# B&R Automation Studio project Lab2_Conveyor (part 4)

### Program Logical/Sorting/AlarmCtrl (IEC) - Alarm control for sorter

#### Cyclic.ld - Cyclic code
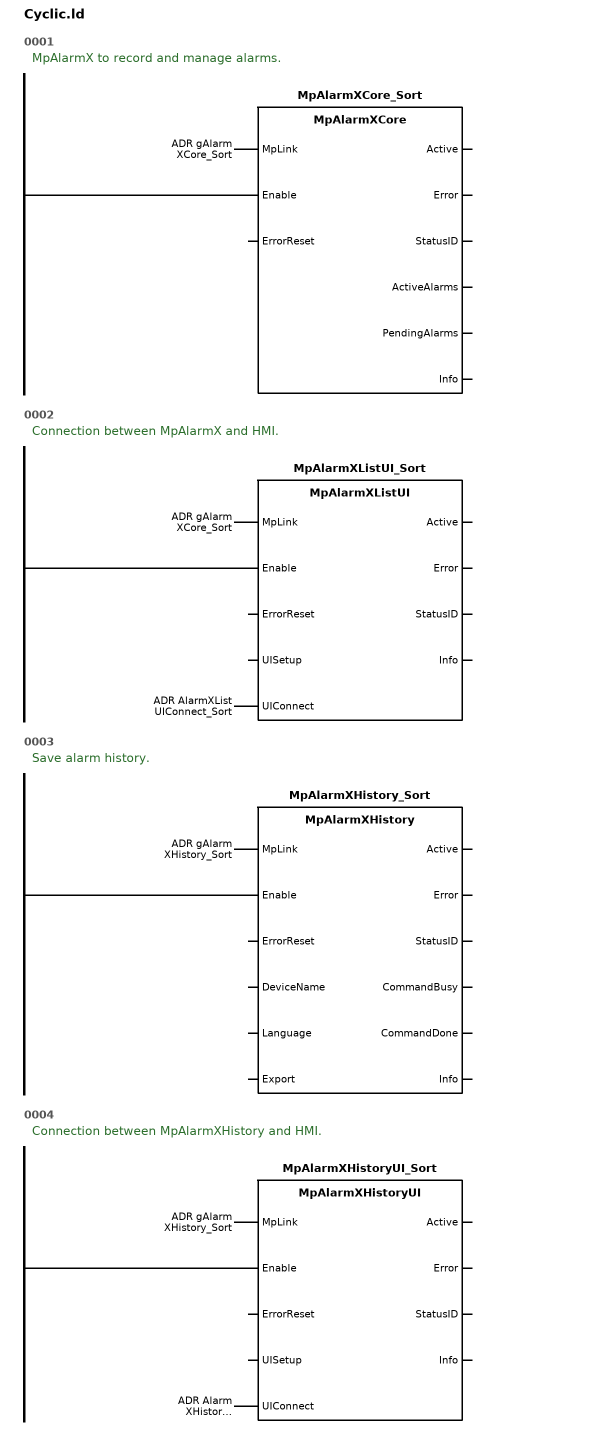
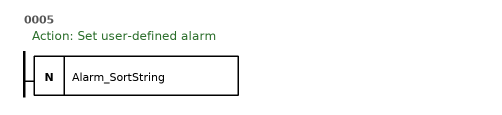
Ladder, written as Structured Text:
```iecst
(*********************************************************************************
 * Copyright: 	Hartfiel Automation
 * Author:    	cashley
 * Created:   	March 8, 2019/12:43 PM
 * Description: 	This file contains alarm handling for the sorting 		station.
 *********************************************************************************)
PROGRAM _CYCLIC
(* Network 1: MpAlarmX to record and manage alarms. *)
MpAlarmXCore_Sort(MpLink := ADR(gAlarmXCore_Sort), Enable := TRUE);

(* Network 2: Connection between MpAlarmX and HMI. *)
MpAlarmXListUI_Sort(MpLink := ADR(gAlarmXCore_Sort), Enable := TRUE, UIConnect := ADR(AlarmXListUIConnect_Sort));

(* Network 3: Save alarm history. *)
MpAlarmXHistory_Sort(MpLink := ADR(gAlarmXHistory_Sort), Enable := TRUE);

(* Network 4: Connection between MpAlarmXHistory and HMI. *)
MpAlarmXHistoryUI_Sort(MpLink := ADR(gAlarmXHistory_Sort), Enable := TRUE, UIConnect := ADR(AlarmXHistoryUIConnect_Sort));

(* Network 5: Action: Set user-defined alarm *)
Alarm_SortString;
END_PROGRAM
```

#### Alarm_SortString.st - Alarm action file
```iecst
(*********************************************************************************
 * Copyright: 	Hartfiel Automation
 * Author:    	cashley
 * Created:   	March 14, 2019/12:00 PM
 * Description: This is an action file that determines the error ID for
				user-defined alarms for the sorting station.
 *********************************************************************************)

ACTION Alarm_SortString:

	//Error ID determines unique name for MpAlarmXSet
	IF Station.Output.Status.ErrorID 	= 1 THEN
		ErrorString := 'Lane1Full';
	ELSIF Station.Output.Status.ErrorID = 2 THEN
		ErrorString := 'Lane2Full';
	ELSIF Station.Output.Status.ErrorID = 3 THEN
		ErrorString := 'Lane3Full';
	ELSIF Station.Output.Status.ErrorID = 4 THEN
		ErrorString := 'NoProductAvail';
	ELSIF Station.Output.Status.ErrorID = 5 THEN
		ErrorString := 'SwitchStuck';
	ELSIF Station.Output.Status.ErrorID = 6 THEN
		ErrorString := 'PuckMissing';
	ELSIF Station.Output.Status.ErrorID = 7 THEN
		ErrorString := 'Axis';
	ELSIF Station.Output.Status.ErrorID = 8 THEN
		ErrorString := 'CheckHW';
	ELSIF Station.Output.Status.ErrorID = 9 THEN
		ErrorString := 'CheckMachine';
	END_IF

	//MpAlarmXSet - enables user-defined alarms
	IF EDGEPOS(Station.Output.Status.Error) THEN
		MpAlarmXSet(MpLink := gAlarmXCore_Sort, Name := ErrorString);
	END_IF

END_ACTION
```

### HwGlobal.typ - not listed in the package file held
```iecst
TYPE
	gSortHW_type : 	STRUCT  (*Hardware IO types for sorter*)
		di : di_type; (*Digital inputs for sorter*)
		do : do_type; (*Digital outputs for sorter*)
	END_STRUCT;
	di_type : 	STRUCT  (*Digital inputs for sorter*)
		ProductAvailable : BOOL; (*Product available*)
		Metallic : BOOL; (*Metallic product*)
		NotBlack : BOOL; (*Product is not black*)
		LaneFull : BOOL; (*Lane full*)
		Switch1Retracted : BOOL; (*Switch 1 retracted*)
		Switch1Extended : BOOL; (*Switch 1 extended*)
		Switch2Retracted : BOOL; (*Switch 2 retracted*)
		Switch2Extended : BOOL; (*Switch 2 extended*)
	END_STRUCT;
	do_type : 	STRUCT  (*Digital outputs for sorter*)
		ExtendSwitch1 : BOOL; (*Extend switch 1*)
		ExtendSwitch2 : BOOL; (*Extend switch 2*)
		RetractStopper : BOOL; (*Retract stopper*)
	END_STRUCT;
END_TYPE
```

### HwGlobal.var - not listed in the package file held
```iecst
VAR
	gSortHW : gSortHW_type; (*Control variable for hardware IO types for sorter*)
END_VAR
```

Listed in the project but not available here: Logical/Global.typ, Logical/acp10etxen, Logical/Distributing/Machine/Conveyor/Conveyor/Init.ld, Logical/Distributing/Machine/Conveyor/Conveyor/Exit.ld, Logical/Distributing/Machine/MainCtrl1/Init.ld, Logical/Distributing/Machine/Ejector/Init.ld, Logical/Distributing/Machine/Ejector/Exit.ld, Logical/Distributing/Machine/Ejector/StateError.ld, Logical/Distributing/Machine/MainCtrl/Init.ld, Logical/Distributing/Machine/MainCtrl/Exit.ld, Logical/Distributing/Machine/SwivelDrive/Init.ld, Logical/Distributing/Machine/SwivelDrive/Exit.ld, Logical/Distributing/Machine/SwivelDrive/StateError.ld, Logical/Distributing/AlarmCtrl/Init.ld, Logical/Distributing/AlarmCtrl/Exit.ld, Logical/Distributing/AlarmCtrl/Types.typ, Logical/Sorting/OPCUA/OPCUA.var, Logical/Sorting/AlarmCtrl/Init.ld, Logical/Sorting/AlarmCtrl/Exit.ld, Logical/Sorting/AlarmCtrl/Types.typ
